// TIA Portal V20 export
ORGANIZATION_BLOCK "Startup"   // OB1020, LAD, Startup
TITLE = "Complete Restart"
// stored: AutoNumber false, IsIECCheckEnabled true, Namespace Unit1.Em3, SetENOAutomatically true
   VAR_INPUT
      LostRetentive : Bool;   // True if retentive data are lost
      LostRTC : Bool;   // True if date and time are lost
   END_VAR
BEGIN

REGION Network 1 (SCL): Build the Absolut Reference Designator
   // Set the Absoult Reference Designator in the Config DB
   IF LEN(IN := "Unit1.Em3.Config".em.referenceDesignator.parent) <> 0 THEN
       "Unit1.Em3.Config".em.referenceDesignator.combined := CONCAT_WSTRING(IN1 := "Unit1.Em3.Config".em.referenceDesignator.parent, IN2 := WSTRING#'.', IN3 := "Unit1.Em3.Config".em.referenceDesignator.relative);
   ELSE
       "Unit1.Em3.Config".em.referenceDesignator.combined := "Unit1.Em3.Config".em.referenceDesignator.relative;
   END_IF;
END_REGION

REGION Network 2 (SCL): Axes data
   // This is an example how to assign axes to DB_ANY in DB Config. If you have axes, assign them here. The Config.axis[] variables will be handed over to the control modules. That enables a flexible programming.
   // // Assign axes
   "Unit1.Em3.Config".axis[1] := "BA060AZSIDR5_TopTapeAxisX";
   "Unit1.Em3.Config".axis[2] := "BA060AZSIDR6_TopTapeAxisY";

   // FB Enable
   "Unit1.Em3.HmiInterface".cmTopTapeAxisX.commands.enableMasterControl := TRUE;
   "Unit1.Em3.HmiInterface".cmTopTapeAxisY.commands.enableMasterControl := TRUE;
END_REGION
END_ORGANIZATION_BLOCK
